TYPE st_driveControl :
STRUCT
	
	xForward		: BOOL;
	xReverse		: BOOL;
	actualposition  : REAL;

END_STRUCT
END_TYPE

(* stored: Version 1.1.0.1, ProductVersion 3.1.4024.12
   DUT st_driveControl: Id {a432210e-a48e-47bc-bccb-e82b09aab905} *)
